FUNCTION_BLOCK ProximitySensor IMPLEMENTS itfReturnBOOL
VAR_INPUT
	ProximityInput : ProxI;
END_VAR
VAR_OUTPUT
END_VAR
VAR
	ProxComp : itfDetectImplement;
	Prox : itfDetect;
END_VAR

Map();

METHOD PRIVATE Map : BOOL
VAR_INPUT
END_VAR
Prox := ProxComp;
Prox.pDetectSignal := ProximityInput.Signal;
END_METHOD

{warning 'add method implementation '}
METHOD mReturnBOOL : BOOL
mReturnBOOL := Prox.pDetectSignal;
END_METHOD

END_FUNCTION_BLOCK

(* stored: Version 1.1.0.1, ProductVersion 3.1.4024.12
   POU ProximitySensor: Id {be2ea9f6-e576-4728-885a-0a0a2bb3dc3a}, SpecialFunc None
   Method Map: Id {dd0a1b0c-8f44-4b93-867d-2b667834846a}
   Method mReturnBOOL: Id {2187815a-a0d5-490d-b1bc-d514041daf77} *)
